# EPICS autosave request: iocs/pvcamIOC/iocBoot/iocPvCam/auto_settings.req
file "pvCam_settings.req",  	    P=$(P),  R=pvcam:
file "NDStdArrays_settings.req",  P=$(P),  R=image1:
file "commonPlugin_settings.req", P=$(P)
